		MoveL OpenholeUD_6675, v10, fine, pHeader\WObj:=wobj0;
		MoveL OpenholeUD_6676, v10, fine, pHeader\WObj:=wobj0;
		MoveL OpenholeUD_6677, v10, fine, pHeader\WObj:=wobj0;
		MoveL OpenholeUD_6678, v10, fine, pHeader\WObj:=wobj0;
		MoveL OpenholeUD_6679, v10, fine, pHeader\WObj:=wobj0;
		MoveL OpenholeUD_6680, v10, fine, pHeader\WObj:=wobj0;
		MoveL OpenholeUD_6681, v10, fine, pHeader\WObj:=wobj0;
		MoveL OpenholeUD_6682, v10, fine, pHeader\WObj:=wobj0;
		MoveL OpenholeUD_6683, v10, fine, pHeader\WObj:=wobj0;
		MoveL OpenholeUD_6684, v10, fine, pHeader\WObj:=wobj0;
		MoveL OpenholeUD_6685, v10, fine, pHeader\WObj:=wobj0;
		MoveL OpenholeUD_6686, v10, fine, pHeader\WObj:=wobj0;
		MoveL OpenholeUD_6687, v10, fine, pHeader\WObj:=wobj0;
		MoveL OpenholeUD_6688, v10, fine, pHeader\WObj:=wobj0;
		MoveL OpenholeUD_6689, v10, fine, pHeader\WObj:=wobj0;
		MoveL OpenholeUD_6690, v10, fine, pHeader\WObj:=wobj0;
		MoveL OpenholeUD_6691, v10, fine, pHeader\WObj:=wobj0;
		MoveL OpenholeUD_6692, v10, fine, pHeader\WObj:=wobj0;
		MoveL OpenholeUD_6693, v10, fine, pHeader\WObj:=wobj0;
		MoveL OpenholeUD_6694, v10, fine, pHeader\WObj:=wobj0;
		MoveL OpenholeUD_6695, v10, fine, pHeader\WObj:=wobj0;
		MoveL OpenholeUD_6696, v10, fine, pHeader\WObj:=wobj0;
		MoveL OpenholeUD_6697, v10, fine, pHeader\WObj:=wobj0;
		MoveL OpenholeUD_6698, v10, fine, pHeader\WObj:=wobj0;
		MoveL OpenholeUD_6699, v10, fine, pHeader\WObj:=wobj0;
		MoveL OpenholeUD_6700, v10, fine, pHeader\WObj:=wobj0;
		MoveL OpenholeUD_6701, v10, fine, pHeader\WObj:=wobj0;
		MoveL OpenholeUD_6702, v10, fine, pHeader\WObj:=wobj0;
		MoveL OpenholeUD_6703, v10, fine, pHeader\WObj:=wobj0;
		MoveL OpenholeUD_6704, v10, fine, pHeader\WObj:=wobj0;
		MoveL OpenholeUD_6705, v10, fine, pHeader\WObj:=wobj0;
		MoveL OpenholeUD_6706, v10, fine, pHeader\WObj:=wobj0;
		MoveL OpenholeUD_6707, v10, fine, pHeader\WObj:=wobj0;
		MoveL OpenholeUD_6708, v10, fine, pHeader\WObj:=wobj0;
		MoveL OpenholeUD_6709, v10, fine, pHeader\WObj:=wobj0;
		MoveL OpenholeUD_6710, v10, fine, pHeader\WObj:=wobj0;
		MoveL OpenholeUD_6711, v10, fine, pHeader\WObj:=wobj0;
		MoveL OpenholeUD_6712, v10, fine, pHeader\WObj:=wobj0;
		MoveL OpenholeUD_6713, v10, fine, pHeader\WObj:=wobj0;
		MoveL OpenholeUD_6714, v10, fine, pHeader\WObj:=wobj0;
		MoveL OpenholeUD_6715, v10, fine, pHeader\WObj:=wobj0;
		MoveL OpenholeUD_6716, v10, fine, pHeader\WObj:=wobj0;
		MoveL OpenholeUD_6717, v10, fine, pHeader\WObj:=wobj0;
		MoveL OpenholeUD_6718, v10, fine, pHeader\WObj:=wobj0;
		MoveL OpenholeUD_6719, v10, fine, pHeader\WObj:=wobj0;
		MoveL OpenholeUD_6720, v10, fine, pHeader\WObj:=wobj0;
		MoveL OpenholeUD_6721, v10, fine, pHeader\WObj:=wobj0;
		MoveL OpenholeUD_6722, v10, fine, pHeader\WObj:=wobj0;
		MoveL OpenholeUD_6723, v10, fine, pHeader\WObj:=wobj0;
		MoveL OpenholeUD_6724, v10, fine, pHeader\WObj:=wobj0;
		MoveL OpenholeUD_6725, v10, fine, pHeader\WObj:=wobj0;
		MoveL OpenholeUD_6726, v10, fine, pHeader\WObj:=wobj0;
		MoveL OpenholeUD_6727, v10, fine, pHeader\WObj:=wobj0;
		MoveL OpenholeUD_6728, v10, fine, pHeader\WObj:=wobj0;
		MoveL OpenholeUD_6729, v10, fine, pHeader\WObj:=wobj0;
		MoveL OpenholeUD_6730, v10, fine, pHeader\WObj:=wobj0;
		MoveL OpenholeUD_6731, v10, fine, pHeader\WObj:=wobj0;
		MoveL OpenholeUD_6732, v10, fine, pHeader\WObj:=wobj0;
		MoveL OpenholeUD_6733, v10, fine, pHeader\WObj:=wobj0;
		MoveL OpenholeUD_6734, v10, fine, pHeader\WObj:=wobj0;
		MoveL OpenholeUD_6735, v10, fine, pHeader\WObj:=wobj0;
		MoveL OpenholeUD_6736, v10, fine, pHeader\WObj:=wobj0;
		MoveL OpenholeUD_6737, v10, fine, pHeader\WObj:=wobj0;
		MoveL OpenholeUD_6738, v10, fine, pHeader\WObj:=wobj0;
		MoveL OpenholeUD_6739, v10, fine, pHeader\WObj:=wobj0;
		MoveL OpenholeUD_6740, v10, fine, pHeader\WObj:=wobj0;
		MoveL OpenholeUD_6741, v10, fine, pHeader\WObj:=wobj0;
		MoveL OpenholeUD_6742, v10, fine, pHeader\WObj:=wobj0;
		MoveL OpenholeUD_6743, v10, fine, pHeader\WObj:=wobj0;
		MoveL OpenholeUD_6744, v10, fine, pHeader\WObj:=wobj0;
		MoveL OpenholeUD_6745, v10, fine, pHeader\WObj:=wobj0;
		MoveL OpenholeUD_6746, v10, fine, pHeader\WObj:=wobj0;
		MoveL OpenholeUD_6747, v10, fine, pHeader\WObj:=wobj0;
		MoveL OpenholeUD_6748, v10, fine, pHeader\WObj:=wobj0;
		MoveL OpenholeUD_6749, v10, fine, pHeader\WObj:=wobj0;
		MoveL OpenholeUD_6750, v10, fine, pHeader\WObj:=wobj0;
		MoveL OpenholeUD_6751, v10, fine, pHeader\WObj:=wobj0;
		MoveL OpenholeUD_6752, v10, fine, pHeader\WObj:=wobj0;
		MoveL OpenholeUD_6753, v10, fine, pHeader\WObj:=wobj0;
		MoveL OpenholeUD_6754, v10, fine, pHeader\WObj:=wobj0;
		MoveL OpenholeUD_6755, v10, fine, pHeader\WObj:=wobj0;
		MoveL OpenholeUD_6756, v10, fine, pHeader\WObj:=wobj0;
		MoveL OpenholeUD_6757, v10, fine, pHeader\WObj:=wobj0;
		MoveL OpenholeUD_6758, v10, fine, pHeader\WObj:=wobj0;
		MoveL OpenholeUD_6759, v10, fine, pHeader\WObj:=wobj0;
		MoveL OpenholeUD_6760, v10, fine, pHeader\WObj:=wobj0;
		MoveL OpenholeUD_6761, v10, fine, pHeader\WObj:=wobj0;
		MoveL OpenholeUD_6762, v10, fine, pHeader\WObj:=wobj0;
		MoveL OpenholeUD_6763, v10, fine, pHeader\WObj:=wobj0;
		MoveL OpenholeUD_6764, v10, fine, pHeader\WObj:=wobj0;
		MoveL OpenholeUD_6765, v10, fine, pHeader\WObj:=wobj0;
		MoveL OpenholeUD_6766, v10, fine, pHeader\WObj:=wobj0;
		MoveL OpenholeUD_6767, v10, fine, pHeader\WObj:=wobj0;
		MoveL OpenholeUD_6768, v10, fine, pHeader\WObj:=wobj0;
		MoveL OpenholeUD_6769, v10, fine, pHeader\WObj:=wobj0;
		MoveL OpenholeUD_6770, v10, fine, pHeader\WObj:=wobj0;
		MoveL OpenholeUD_6771, v10, fine, pHeader\WObj:=wobj0;
		MoveL OpenholeUD_6772, v10, fine, pHeader\WObj:=wobj0;
		MoveL OpenholeUD_6773, v10, fine, pHeader\WObj:=wobj0;
		MoveL OpenholeUD_6774, v10, fine, pHeader\WObj:=wobj0;
		MoveL OpenholeUD_6775, v10, fine, pHeader\WObj:=wobj0;
		MoveL OpenholeUD_6776, v10, fine, pHeader\WObj:=wobj0;
		MoveL OpenholeUD_6777, v10, fine, pHeader\WObj:=wobj0;
		MoveL OpenholeUD_6778, v10, fine, pHeader\WObj:=wobj0;
		MoveL OpenholeUD_6779, v10, fine, pHeader\WObj:=wobj0;
		MoveL OpenholeUD_6780, v10, fine, pHeader\WObj:=wobj0;
		MoveL OpenholeUD_6781, v10, fine, pHeader\WObj:=wobj0;
		MoveL OpenholeUD_6782, v10, fine, pHeader\WObj:=wobj0;
		MoveL OpenholeUD_6783, v10, fine, pHeader\WObj:=wobj0;
		MoveL OpenholeUD_6784, v10, fine, pHeader\WObj:=wobj0;
		MoveL OpenholeUD_6785, v10, fine, pHeader\WObj:=wobj0;
		MoveL OpenholeUD_6786, v10, fine, pHeader\WObj:=wobj0;
		MoveL OpenholeUD_6787, v10, fine, pHeader\WObj:=wobj0;
		MoveL OpenholeUD_6788, v10, fine, pHeader\WObj:=wobj0;
		MoveL OpenholeUD_6789, v10, fine, pHeader\WObj:=wobj0;
		MoveL OpenholeUD_6790, v10, fine, pHeader\WObj:=wobj0;
		MoveL OpenholeUD_6791, v10, fine, pHeader\WObj:=wobj0;
		MoveL OpenholeUD_6792, v10, fine, pHeader\WObj:=wobj0;
		MoveL OpenholeUD_6793, v10, fine, pHeader\WObj:=wobj0;
		MoveL OpenholeUD_6794, v10, fine, pHeader\WObj:=wobj0;
		MoveL OpenholeUD_6795, v10, fine, pHeader\WObj:=wobj0;
		MoveL OpenholeUD_6796, v10, fine, pHeader\WObj:=wobj0;
		MoveL OpenholeUD_6797, v10, fine, pHeader\WObj:=wobj0;
		MoveL OpenholeUD_6798, v10, fine, pHeader\WObj:=wobj0;
		MoveL OpenholeUD_6799, v10, fine, pHeader\WObj:=wobj0;
		MoveL OpenholeUD_6800, v10, fine, pHeader\WObj:=wobj0;
		MoveL OpenholeUD_6801, v10, fine, pHeader\WObj:=wobj0;
		MoveL OpenholeUD_6802, v10, fine, pHeader\WObj:=wobj0;
		MoveL OpenholeUD_6803, v10, fine, pHeader\WObj:=wobj0;
		MoveL OpenholeUD_6804, v10, fine, pHeader\WObj:=wobj0;
		MoveL OpenholeUD_6805, v10, fine, pHeader\WObj:=wobj0;
		MoveL OpenholeUD_6806, v10, fine, pHeader\WObj:=wobj0;
		MoveL OpenholeUD_6807, v10, fine, pHeader\WObj:=wobj0;
		MoveL OpenholeUD_6808, v10, fine, pHeader\WObj:=wobj0;
		MoveL OpenholeUD_6809, v10, fine, pHeader\WObj:=wobj0;
		MoveL OpenholeUD_6810, v10, fine, pHeader\WObj:=wobj0;
		MoveL OpenholeUD_6811, v10, fine, pHeader\WObj:=wobj0;
		MoveL OpenholeUD_6812, v10, fine, pHeader\WObj:=wobj0;
		MoveL OpenholeUD_6813, v10, fine, pHeader\WObj:=wobj0;
		MoveL OpenholeUD_6814, v10, fine, pHeader\WObj:=wobj0;
		MoveL OpenholeUD_6815, v10, fine, pHeader\WObj:=wobj0;
		MoveL OpenholeUD_6816, v10, fine, pHeader\WObj:=wobj0;
		MoveL OpenholeUD_6817, v10, fine, pHeader\WObj:=wobj0;
		MoveL OpenholeUD_6818, v10, fine, pHeader\WObj:=wobj0;
		MoveL OpenholeUD_6819, v10, fine, pHeader\WObj:=wobj0;
		MoveL OpenholeUD_6820, v10, fine, pHeader\WObj:=wobj0;
		MoveL OpenholeUD_6821, v10, fine, pHeader\WObj:=wobj0;
		MoveL OpenholeUD_6822, v10, fine, pHeader\WObj:=wobj0;
		MoveL OpenholeUD_6823, v10, fine, pHeader\WObj:=wobj0;
		MoveL OpenholeUD_6824, v10, fine, pHeader\WObj:=wobj0;
		MoveL OpenholeUD_6825, v10, fine, pHeader\WObj:=wobj0;
		MoveL OpenholeUD_6826, v10, fine, pHeader\WObj:=wobj0;
		MoveL OpenholeUD_6827, v10, fine, pHeader\WObj:=wobj0;
		MoveL OpenholeUD_6828, v10, fine, pHeader\WObj:=wobj0;
		MoveL OpenholeUD_6829, v10, fine, pHeader\WObj:=wobj0;
		MoveL OpenholeUD_6830, v10, fine, pHeader\WObj:=wobj0;
		MoveL OpenholeUD_6831, v10, fine, pHeader\WObj:=wobj0;
		MoveL OpenholeUD_6832, v10, fine, pHeader\WObj:=wobj0;
		MoveL OpenholeUD_6833, v10, fine, pHeader\WObj:=wobj0;
		MoveL OpenholeUD_6834, v10, fine, pHeader\WObj:=wobj0;
		MoveL OpenholeUD_6835, v10, fine, pHeader\WObj:=wobj0;
		MoveL OpenholeUD_6836, v10, fine, pHeader\WObj:=wobj0;
		MoveL OpenholeUD_6837, v10, fine, pHeader\WObj:=wobj0;
		MoveL OpenholeUD_6838, v10, fine, pHeader\WObj:=wobj0;
		MoveL OpenholeUD_6839, v10, fine, pHeader\WObj:=wobj0;
		MoveL OpenholeUD_6840, v10, fine, pHeader\WObj:=wobj0;
		MoveL OpenholeUD_6841, v10, fine, pHeader\WObj:=wobj0;
		MoveL OpenholeUD_6842, v10, fine, pHeader\WObj:=wobj0;
		MoveL OpenholeUD_6843, v10, fine, pHeader\WObj:=wobj0;
		MoveL OpenholeUD_6844, v10, fine, pHeader\WObj:=wobj0;
		MoveL OpenholeUD_6845, v10, fine, pHeader\WObj:=wobj0;
		MoveL OpenholeUD_6846, v10, fine, pHeader\WObj:=wobj0;
		MoveL OpenholeUD_6847, v10, fine, pHeader\WObj:=wobj0;
		MoveL OpenholeUD_6848, v10, fine, pHeader\WObj:=wobj0;
		MoveL OpenholeUD_6849, v10, fine, pHeader\WObj:=wobj0;
		MoveL OpenholeUD_6850, v10, fine, pHeader\WObj:=wobj0;
		MoveL OpenholeUD_6851, v10, fine, pHeader\WObj:=wobj0;
		MoveL OpenholeUD_6852, v10, fine, pHeader\WObj:=wobj0;
		MoveL OpenholeUD_6853, v10, fine, pHeader\WObj:=wobj0;
		MoveL OpenholeUD_6854, v10, fine, pHeader\WObj:=wobj0;
		MoveL OpenholeUD_6855, v10, fine, pHeader\WObj:=wobj0;
		MoveL OpenholeUD_6856, v10, fine, pHeader\WObj:=wobj0;
		MoveL OpenholeUD_6857, v10, fine, pHeader\WObj:=wobj0;
		MoveL OpenholeUD_6858, v10, fine, pHeader\WObj:=wobj0;
		MoveL OpenholeUD_6859, v10, fine, pHeader\WObj:=wobj0;
		MoveL OpenholeUD_6860, v10, fine, pHeader\WObj:=wobj0;
		MoveL OpenholeUD_6861, v10, fine, pHeader\WObj:=wobj0;
		MoveL OpenholeUD_6862, v10, fine, pHeader\WObj:=wobj0;
		MoveL OpenholeUD_6863, v10, fine, pHeader\WObj:=wobj0;
		MoveL OpenholeUD_6864, v10, fine, pHeader\WObj:=wobj0;
		MoveL OpenholeUD_6865, v10, fine, pHeader\WObj:=wobj0;
		MoveL OpenholeUD_6866, v10, fine, pHeader\WObj:=wobj0;
		MoveL OpenholeUD_6867, v10, fine, pHeader\WObj:=wobj0;
		MoveL OpenholeUD_6868, v10, fine, pHeader\WObj:=wobj0;
		MoveL OpenholeUD_6869, v10, fine, pHeader\WObj:=wobj0;
		MoveL OpenholeUD_6870, v10, fine, pHeader\WObj:=wobj0;
		MoveL OpenholeUD_6871, v10, fine, pHeader\WObj:=wobj0;
		MoveL OpenholeUD_6872, v10, fine, pHeader\WObj:=wobj0;
		MoveL OpenholeUD_6873, v10, fine, pHeader\WObj:=wobj0;
		MoveL OpenholeUD_6874, v10, fine, pHeader\WObj:=wobj0;
		MoveL OpenholeUD_6875, v10, fine, pHeader\WObj:=wobj0;
		MoveL OpenholeUD_6876, v10, fine, pHeader\WObj:=wobj0;
		MoveL OpenholeUD_6877, v10, fine, pHeader\WObj:=wobj0;
		MoveL OpenholeUD_6878, v10, fine, pHeader\WObj:=wobj0;
		MoveL OpenholeUD_6879, v10, fine, pHeader\WObj:=wobj0;
		MoveL OpenholeUD_6880, v10, fine, pHeader\WObj:=wobj0;
		MoveL OpenholeUD_6881, v10, fine, pHeader\WObj:=wobj0;
		MoveL OpenholeUD_6882, v10, fine, pHeader\WObj:=wobj0;
		MoveL OpenholeUD_6883, v10, fine, pHeader\WObj:=wobj0;
		MoveL OpenholeUD_6884, v10, fine, pHeader\WObj:=wobj0;
		MoveL OpenholeUD_6885, v10, fine, pHeader\WObj:=wobj0;
		MoveL OpenholeUD_6886, v10, fine, pHeader\WObj:=wobj0;
		MoveL OpenholeUD_6887, v10, fine, pHeader\WObj:=wobj0;
		MoveL OpenholeUD_6888, v10, fine, pHeader\WObj:=wobj0;
		MoveL OpenholeUD_6889, v10, fine, pHeader\WObj:=wobj0;
		MoveL OpenholeUD_6890, v10, fine, pHeader\WObj:=wobj0;
		MoveL OpenholeUD_6891, v10, fine, pHeader\WObj:=wobj0;
		MoveL OpenholeUD_6892, v10, fine, pHeader\WObj:=wobj0;
		MoveL OpenholeUD_6893, v10, fine, pHeader\WObj:=wobj0;
		MoveL OpenholeUD_6894, v10, fine, pHeader\WObj:=wobj0;
		MoveL OpenholeUD_6895, v10, fine, pHeader\WObj:=wobj0;
		MoveL OpenholeUD_6896, v10, fine, pHeader\WObj:=wobj0;
		MoveL OpenholeUD_6897, v10, fine, pHeader\WObj:=wobj0;
		MoveL OpenholeUD_6898, v10, fine, pHeader\WObj:=wobj0;
		MoveL OpenholeUD_6899, v10, fine, pHeader\WObj:=wobj0;
		MoveL OpenholeUD_6900, v10, fine, pHeader\WObj:=wobj0;
		MoveL OpenholeUD_6901, v10, fine, pHeader\WObj:=wobj0;
		MoveL OpenholeUD_6902, v10, fine, pHeader\WObj:=wobj0;
		MoveL OpenholeUD_6903, v10, fine, pHeader\WObj:=wobj0;
		MoveL OpenholeUD_6904, v10, fine, pHeader\WObj:=wobj0;
		MoveL OpenholeUD_6905, v10, fine, pHeader\WObj:=wobj0;
		MoveL OpenholeUD_6906, v10, fine, pHeader\WObj:=wobj0;
		MoveL OpenholeUD_6907, v10, fine, pHeader\WObj:=wobj0;
		MoveL OpenholeUD_6908, v10, fine, pHeader\WObj:=wobj0;
		MoveL OpenholeUD_6909, v10, fine, pHeader\WObj:=wobj0;
		MoveL OpenholeUD_6910, v10, fine, pHeader\WObj:=wobj0;
		MoveL OpenholeUD_6911, v10, fine, pHeader\WObj:=wobj0;
		MoveL OpenholeUD_6912, v10, fine, pHeader\WObj:=wobj0;
		MoveL OpenholeUD_6913, v10, fine, pHeader\WObj:=wobj0;
		MoveL OpenholeUD_6914, v10, fine, pHeader\WObj:=wobj0;
		MoveL OpenholeUD_6915, v10, fine, pHeader\WObj:=wobj0;
		MoveL OpenholeUD_6916, v10, fine, pHeader\WObj:=wobj0;
		MoveL OpenholeUD_6917, v10, fine, pHeader\WObj:=wobj0;
		MoveL OpenholeUD_6918, v10, fine, pHeader\WObj:=wobj0;
		MoveL OpenholeUD_6919, v10, fine, pHeader\WObj:=wobj0;
		MoveL OpenholeUD_6920, v10, fine, pHeader\WObj:=wobj0;
		MoveL OpenholeUD_6921, v10, fine, pHeader\WObj:=wobj0;
		MoveL OpenholeUD_6922, v10, fine, pHeader\WObj:=wobj0;
		MoveL OpenholeUD_6923, v10, fine, pHeader\WObj:=wobj0;
		MoveL OpenholeUD_6924, v10, fine, pHeader\WObj:=wobj0;
		MoveL OpenholeUD_6925, v10, fine, pHeader\WObj:=wobj0;
		MoveL OpenholeUD_6926, v10, fine, pHeader\WObj:=wobj0;
		MoveL OpenholeUD_6927, v10, fine, pHeader\WObj:=wobj0;
		MoveL OpenholeUD_6928, v10, fine, pHeader\WObj:=wobj0;
		MoveL OpenholeUD_6929, v10, fine, pHeader\WObj:=wobj0;
		MoveL OpenholeUD_6930, v10, fine, pHeader\WObj:=wobj0;
		MoveL OpenholeUD_6931, v10, fine, pHeader\WObj:=wobj0;
		MoveL OpenholeUD_6932, v10, fine, pHeader\WObj:=wobj0;
		MoveL OpenholeUD_6933, v10, fine, pHeader\WObj:=wobj0;
		MoveL OpenholeUD_6934, v10, fine, pHeader\WObj:=wobj0;
		MoveL OpenholeUD_6935, v10, fine, pHeader\WObj:=wobj0;
		MoveL OpenholeUD_6936, v10, fine, pHeader\WObj:=wobj0;
		MoveL OpenholeUD_6937, v10, fine, pHeader\WObj:=wobj0;
		MoveL OpenholeUD_6938, v10, fine, pHeader\WObj:=wobj0;
		MoveL OpenholeUD_6939, v10, fine, pHeader\WObj:=wobj0;
		MoveL OpenholeUD_6940, v10, fine, pHeader\WObj:=wobj0;
		MoveL OpenholeUD_6941, v10, fine, pHeader\WObj:=wobj0;
		MoveL OpenholeUD_6942, v10, fine, pHeader\WObj:=wobj0;
		MoveL OpenholeUD_6943, v10, fine, pHeader\WObj:=wobj0;
		MoveL OpenholeUD_6944, v10, fine, pHeader\WObj:=wobj0;
		MoveL OpenholeUD_6945, v10, fine, pHeader\WObj:=wobj0;
		MoveL OpenholeUD_6946, v10, fine, pHeader\WObj:=wobj0;
		MoveL OpenholeUD_6947, v10, fine, pHeader\WObj:=wobj0;
		MoveL OpenholeUD_6948, v10, fine, pHeader\WObj:=wobj0;
		MoveL OpenholeUD_6949, v10, fine, pHeader\WObj:=wobj0;
		MoveL OpenholeUD_6950, v10, fine, pHeader\WObj:=wobj0;
		MoveL OpenholeUD_6951, v10, fine, pHeader\WObj:=wobj0;
		MoveL OpenholeUD_6952, v10, fine, pHeader\WObj:=wobj0;
		MoveL OpenholeUD_6953, v10, fine, pHeader\WObj:=wobj0;
		MoveL OpenholeUD_6954, v10, fine, pHeader\WObj:=wobj0;
		MoveL OpenholeUD_6955, v10, fine, pHeader\WObj:=wobj0;
		MoveL OpenholeUD_6956, v10, fine, pHeader\WObj:=wobj0;
		MoveL OpenholeUD_6957, v10, fine, pHeader\WObj:=wobj0;
		MoveL OpenholeUD_6958, v10, fine, pHeader\WObj:=wobj0;
		MoveL OpenholeUD_6959, v10, fine, pHeader\WObj:=wobj0;
		MoveL OpenholeUD_6960, v10, fine, pHeader\WObj:=wobj0;
		MoveL OpenholeUD_6961, v10, fine, pHeader\WObj:=wobj0;
		MoveL OpenholeUD_6962, v10, fine, pHeader\WObj:=wobj0;
		MoveL OpenholeUD_6963, v10, fine, pHeader\WObj:=wobj0;
		MoveL OpenholeUD_6964, v10, fine, pHeader\WObj:=wobj0;
		MoveL OpenholeUD_6965, v10, fine, pHeader\WObj:=wobj0;
		MoveL OpenholeUD_6966, v10, fine, pHeader\WObj:=wobj0;
		MoveL OpenholeUD_6967, v10, fine, pHeader\WObj:=wobj0;
		MoveL OpenholeUD_6968, v10, fine, pHeader\WObj:=wobj0;
		MoveL OpenholeUD_6969, v10, fine, pHeader\WObj:=wobj0;
		MoveL OpenholeUD_6970, v10, fine, pHeader\WObj:=wobj0;
		MoveL OpenholeUD_6971, v10, fine, pHeader\WObj:=wobj0;
		MoveL OpenholeUD_6972, v10, fine, pHeader\WObj:=wobj0;
		MoveL OpenholeUD_6973, v10, fine, pHeader\WObj:=wobj0;
		MoveL OpenholeUD_6974, v10, fine, pHeader\WObj:=wobj0;
		MoveL OpenholeUD_6975, v10, fine, pHeader\WObj:=wobj0;
		MoveL OpenholeUD_6976, v10, fine, pHeader\WObj:=wobj0;
		MoveL OpenholeUD_6977, v10, fine, pHeader\WObj:=wobj0;
		MoveL OpenholeUD_6978, v10, fine, pHeader\WObj:=wobj0;
		MoveL OpenholeUD_6979, v10, fine, pHeader\WObj:=wobj0;
		MoveL OpenholeUD_6980, v10, fine, pHeader\WObj:=wobj0;
		MoveL OpenholeUD_6981, v10, fine, pHeader\WObj:=wobj0;
		MoveL OpenholeUD_6982, v10, fine, pHeader\WObj:=wobj0;
		MoveL OpenholeUD_6983, v10, fine, pHeader\WObj:=wobj0;
	ENDPROC

ENDMODULE
